# EPICS alarm handler configuration: mps_database/bare/alarms/areas/mpln_undh_mp11.alhConfig
GROUP NULL MPLN:UNDH:MP11:1
$ALIAS MPS Link Node 147
$GUIDANCE
LTUH MPS
   Group Name: MPLN:UNDH:MP11:1
   Summary PV:  MPLN:UNDH:MP11:1:STATSUMY
$END
CHANNEL  MPLN:UNDH:MP11:1    MPLN:UNDH:MP11:1:MPS_EN_RBV		-----
CHANNEL  MPLN:UNDH:MP11:1    MPLN:UNDH:MP11:1:LC1_MODE_RBV		-----
